// TIA Portal project "SeniorProject" (V15.1)

(* hardware
DEVICE "S71500/ET200MP station_1"  S7-1500 station
   slot 0: "Rail_0"  Rack  6ES7 590-1***0-0AA0
   slot 1: "PLC_1"  CPU 1511F-1 PN  6ES7 511-1FK02-0AB0  V2.6
      slot 3: "CPU display_1"  6ES7591-1AA00-0AA0
   slot 2: "DI 16x24VDC SRC BA_1"  DI 16x24VDC SRC BA  6ES7 521-1BH50-0AA0  V2.0
   slot 3: "DQ 16x24VDC/0.5A HF_1"  DQ 16x24VDC/0.5A HF  6ES7 522-1BH01-0AB0  V1.0
   slot 4: "F-DI 16x24V DC_1"  F-DI 16x24V DC  6ES7 526-1BH00-0AB0  V1.0
      slot 1: "F-DI 16x24V DC_1"  F-DI 16x24V DC
DEVICE "SINAMICS G_1"  Sinamics.Device
   slot 0: "	_0"  Rail  SinamicsG120RackPN
   slot 0: "G120_CU240E_2_PN"  G120 CU240E-2 PN  6SL3244-0BB12-1FA0  4.5
      slot 1: "PROFINET interface"  MDD-SinamicsG120-P
   slot 3: "PM240 IP20"  PM240 IP20  6SL3224-0BE13-7UA0  -
*)

// ===== PLC "PLC_1"  CPU 1511F-1 PN =====
// protected blocks, not shown: "Main_Safety_RTG1", "Main_Safety_RTG1_DB"

ORGANIZATION_BLOCK "Main"   // OB1, LAD, ProgramCycle
TITLE = "Main Program Sweep (Cycle)"
{ S7_Optimized_Access := 'TRUE' }
VERSION : 0.1
   VAR_INPUT
      Initial_Call : Bool;   // Initial call of this OB
      Remanence : Bool;   // =True, if remanent data are available
   END_VAR
BEGIN
END_ORGANIZATION_BLOCK